{attribute 'pack_mode' := '1'}
TYPE TPearlsArea :
STRUCT
	iNbOfPearls		: INT;
	iFirstPearl		: INT;
END_STRUCT
END_TYPE

(* stored: Version 1.1.0.1, ProductVersion 3.1.4022.12
   DUT TPearlsArea: Id {38bad39b-39c8-4ce4-989f-c52946b04e89} *)
